// TIA Portal V16 export
// export: Created 2023-10-30T22:43:52.2946173Z, ExportSetting WithDefaults, DisplayName Totally Integrated Automation Portal, DisplayVersion V16, DisplayName TIA Portal Version Control Interface, DisplayVersion V16, DisplayName TIA Portal Openness, DisplayVersion V16, DisplayName SINAMICS Startdrive Advanced, DisplayVersion V16, DisplayName SINAMICS Startdrive G130, G150, S120, S150, SINAMICS MV, S210, DisplayVersion V16, DisplayName SINAMICS Startdrive G110M, G120, G120C, G120D, G120P, DisplayVersion V16, DisplayName STEP 7 Professional, DisplayVersion V16, DisplayName STEP 7 Safety, DisplayVersion V16, DisplayName WinCC Professional, DisplayVersion V16
DATA_BLOCK "IEC_Timer_0_DB_6"   // DB29
{ S7_Optimized_Access := 'TRUE' }
// stored: AutoNumber true, DBAccessibleFromOPCUA true, InstanceOfName IEC_TIMER, OfSystemLibElement IEC_TIMER, OfSystemLibVersion 1.0
"IEC_TIMER"
   // VAR
   //    PT : Time;
   //    ET { ExternalWritable := 'False'} : Time;
   //    IN : Bool;
   //    Q { ExternalWritable := 'False'} : Bool;
   // END_VAR
BEGIN
END_DATA_BLOCK
